{attribute addProperty BoxType "EL3783-0000-0018"}
{attribute addProperty Id "U2_SamplesAT %I*ARRAY [0..19] OF INT32040"}
{attribute addProperty CRC "339589939"}
{attribute addProperty SizeInBites "320"}
{attribute addProperty SizeInBytes "40"}
TYPE L2_Voltage_Samples_143DBB33 :
STRUCT
	{attribute addProperty Name "U2_Samples"}
	U2_Samples AT %I* : ARRAY [0..19] OF INT;
END_STRUCT
END_TYPE

(* stored: Version 1.2.0.0, ProductVersion 3.1.4024.9
   DUT L2_Voltage_Samples_143DBB33: Id {ba282053-e5b5-48b7-87c2-1ad1f1d3ad1e} *)
